{attribute 'linkalways'}
{attribute 'hide_all_locals'}
FUNCTION_BLOCK ValueWord EXTENDS ValueWordRead IMPLEMENTS Value
VAR
END_VAR

METHOD SetFromType : BOOL
VAR_INPUT
	source : __SYSTEM.AnyType;
END_VAR
SetFromType := ConvertAnyType(source, thisAnyType);
END_METHOD

METHOD SetFromString : BOOL
VAR_INPUT
	value : T_MaxString;
END_VAR
thisValue := STRING_TO_WORD(value);

SetFromString := TRUE;
END_METHOD

METHOD Set : BOOL
VAR_INPUT
	source : ANY;
END_VAR
Set := ConvertAnyType(source, thisAnyType);
END_METHOD

END_FUNCTION_BLOCK

(* stored: Version 1.1.0.1
   POU ValueWord: Id {66db54ce-c733-4278-b057-96198b259a5c}, SpecialFunc None
   Method SetFromType: Id {2531c687-0113-406f-92eb-843dad21d908}
   Method SetFromString: Id {a8d33874-51bf-4f6e-9463-91ed48d5b273}
   Method Set: Id {231ff19c-9fbb-4340-a67b-e2ed933f2339} *)
